// TIA Portal project "SCL EJERCICIO 3" (V11)

(* hardware
DEVICE "S7300/ET200 station_1"  SIMATIC 300-Station
   slot 0: "Perfil soporte_0"  Rail  6ES7 390-1***0-0AA0
   slot 2: "PLC_1"  CPU 313C-2 DP  6ES7 313-6CF03-0AB0  V2.6
      slot 0: "Interfaz MPI_1"  MPI
      slot 1: "Interfaz DP_1"  DP
      slot 2: "DI16/DO16_1"  DI16/DO16
      slot 4: "Contaje_1"  Counter
*)

// ===== PLC "PLC_1"  CPU 313C-2 DP =====

VAR_GLOBAL   // PLC tag table "Tabla de variables estándar"
   "Tag_1" AT %E0.0 : Bool;
   "Tag_2" AT %E0.1 : Bool;
   "Tag_3" AT %A0.0 : Bool;
   "Tag_4" AT %A0.1 : Bool;
   "Tag_5" AT %A0.2 : Bool;
   "Tag_6" AT %T0 : Timer;
   "Tag_7" AT %E0.2 : Bool;
   "Tag_8" AT %A0.3 : Bool;
   "Tag_9" AT %A0.4 : Bool;
   "Tag_10" AT %A0.5 : Bool;
END_VAR

DATA_BLOCK "Bloque_1_DB"   // DB2
{ S7_Optimized_Access := 'FALSE' }
VERSION : 0.1
// stored: InstanceOfName Bloque_1
"Bloque_1"
BEGIN
END_DATA_BLOCK

FUNCTION_BLOCK "Bloque_1"   // FB1, SCL
{ S7_Optimized_Access := 'FALSE' }
VERSION : 0.1
   VAR_INPUT
      MARCHA : Bool;
      PARO : Bool;
      "RELE TERMICO" : Bool;
   END_VAR
   VAR_OUTPUT
      LINEA : Bool;
      ESTRELLA : Bool;
      TRIANGULO : Bool;
      "LED MARCHA" : Bool;
      "LED PARO" : Bool;
      "LED AVERIA" : Bool;
   END_VAR
   VAR
      VISUALIZAR : Time;
      T0 : Bool;
   END_VAR
BEGIN
   IF #PARO THEN (* cuando esta activada no se podra arrancar el motor y estara encendida led paro *)
     #LINEA:=FALSE;
     #ESTRELLA:=FALSE;
     #TRIANGULO:=FALSE;
     #"LED PARO":=TRUE;
     #"LED MARCHA":=FALSE;
     RETURN;
   END_IF;

   IF  NOT  #LINEA AND NOT #ESTRELLA AND NOT #TRIANGULO AND NOT #"LED MARCHA" THEN(* en reposo led paro encendida *)
       #"LED PARO" := TRUE;
     END_IF;

   IF #MARCHA THEN (* arranca linea y led marcha *)
     #LINEA:=TRUE;
     #"LED MARCHA":=TRUE;
     #"LED PARO":=FALSE;
   END_IF;

   IF #LINEA THEN (* cuando entra liinea conrecta estrella *)
     #ESTRELLA:=TRUE;
   END_IF;

   "IEC_Timer_0_DB".TON(IN:=#LINEA,(*temporizado 3 s *)
                        PT:=T#4S,
                        Q=> #T0,
                        ET=>#VISUALIZAR);


   IF #LINEA AND #T0 THEN (*cambio de conexion desconecta estrella *)
   #ESTRELLA:= FALSE;
     END_IF;

   IF #LINEA AND #T0 THEN (*cambia a triangulo *)
   #TRIANGULO:= TRUE;
   END_IF;

   IF #"RELE TERMICO" THEN (* disparo termico desconecta todo y enciende led de averia mientras este activado y led de paro ,bloquea arranque *)
     #LINEA:=FALSE;
     #ESTRELLA:=FALSE;
     #TRIANGULO:=FALSE;
     #"LED MARCHA":=FALSE;
     #"LED AVERIA":=TRUE;
     #"LED PARO":=TRUE;
   ELSE
     #"LED AVERIA":=FALSE;
     END_IF;
END_FUNCTION_BLOCK

ORGANIZATION_BLOCK "Main"   // OB1, LAD
TITLE = "Main Program Sweep (Cycle)"
{ S7_Optimized_Access := 'FALSE' }
VERSION : 0.1
   VAR_TEMP
      OB1_EV_CLASS : Byte;   // Bits 0-3 = 1 (Coming event), Bits 4-7 = 1 (Event class 1)
      OB1_SCAN_1 : Byte;   // 1 (Cold restart scan 1 of OB 1), 3 (Scan 2-n of OB 1)
      OB1_PRIORITY : Byte;   // Priority of OB Execution
      OB1_OB_NUMBR : Byte;   // 1 (Organization block 1, OB1)
      OB1_RESERVED_1 : Byte;   // Reserved for system
      OB1_RESERVED_2 : Byte;   // Reserved for system
      OB1_PREV_CYCLE : Int;   // Cycle time of previous OB1 scan (milliseconds)
      OB1_MIN_CYCLE : Int;   // Minimum cycle time of OB1 (milliseconds)
      OB1_MAX_CYCLE : Int;   // Maximum cycle time of OB1 (milliseconds)
      OB1_DATE_TIME : Date_And_Time;   // Date and time OB1 started
   END_VAR
BEGIN

REGION Network 1
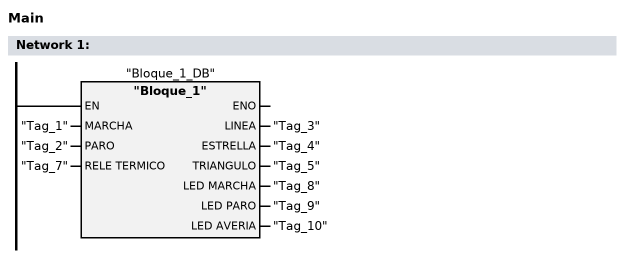
   RUNG wire#powerrail
      "Bloque_1_DB"(MARCHA := "Tag_1", PARO := "Tag_2", "RELE TERMICO" := "Tag_7", LINEA => "Tag_3", ESTRELLA => "Tag_4", TRIANGULO => "Tag_5", "LED MARCHA" => "Tag_8", "LED PARO" => "Tag_9", "LED AVERIA" => "Tag_10")
   END_RUNG
   // the same network as SCL:
   "Bloque_1_DB"(MARCHA := "Tag_1",   // "Bloque_1"
                 PARO := "Tag_2",
                 "RELE TERMICO" := "Tag_7",
                 LINEA => "Tag_3",
                 ESTRELLA => "Tag_4",
                 TRIANGULO => "Tag_5",
                 "LED MARCHA" => "Tag_8",
                 "LED PARO" => "Tag_9",
                 "LED AVERIA" => "Tag_10");
END_REGION
END_ORGANIZATION_BLOCK